{attribute 'linkalways'} 
{attribute 'no_explicit_call' := 'This FB is a CLASS and must be accessed using methods or properties'}
{attribute 'enable_dynamic_creation'}
FUNCTION_BLOCK Node_RGBA_RED EXTENDS VisionNode
VAR
    out : _TcVnVector4_LREAL;
END_VAR

METHOD PUBLIC  Clone : I_Node
VAR
	pNode : POINTER TO Node_RGBA_RED;
END_VAR
pNode := __NEW(Node_RGBA_RED);
Clone := pNode^;
END_METHOD

METHOD FB_init : BOOL
VAR_INPUT
	bInitRetains : BOOL; // if TRUE, the retain variables are initialized (warm start / cold start)
	bInCopyCode : BOOL;  // if TRUE, the instance afterwards gets moved into the copy code (online change)
END_VAR
AddOutput('out', out);
END_METHOD

METHOD PROTECTED OnExecute
out.Value := GVL_COLOURS.RGBA_RED;
END_METHOD

METHOD PUBLIC PreExecutionCheck
VAR_INPUT
	Check : I_PreExecutionChecks;
END_VAR
END_METHOD

END_FUNCTION_BLOCK

(* stored: Version 1.1.0.1, ProductVersion 3.1.4024.13
   POU Node_RGBA_RED: Id {61acc737-2976-09f8-0f80-0f537dc5c537}, SpecialFunc None
   Folder Constructor: Id {09096e0a-d6ac-0035-28b0-265f1dbd6f5b}
   Method Clone: Id {ebf22eeb-1920-07f4-2489-6a6dd52b5037}
   Method FB_init: Id {450a1026-8a34-0067-1cac-ba93e85bf184}
   Method OnExecute: Id {a747307d-ac4b-0735-2225-a17d18ed061c}
   Method PreExecutionCheck: Id {9ac8f97c-f128-0b57-2a12-b6d60bc44554} *)
